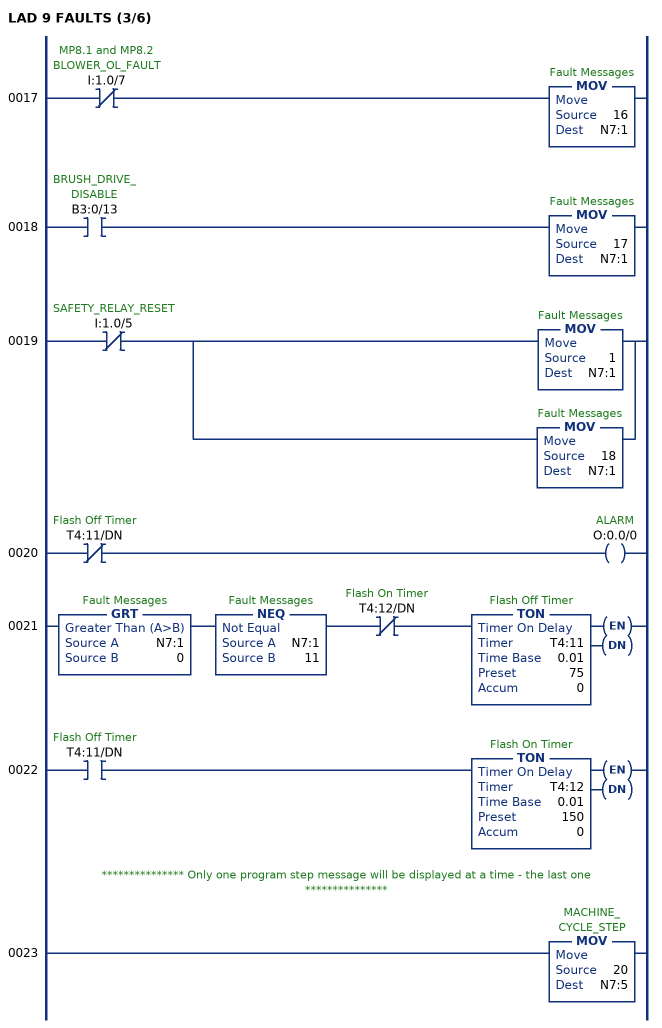
% Rung: 17 %
SOR XIO I:1.0/7 MOV 16 N7:1 EOR
%   I:1.0/7  BLOWER_OL_FAULT  "MP8.1 and MP8.2" %
%   N7:1  "Fault Messages" %
% Rung: 18 %
SOR XIC B3:0/13 MOV 17 N7:1 EOR
%   B3:0/13  BRUSH_DRIVE_DISABLE %
%   N7:1  "Fault Messages" %
% Rung: 19 %
SOR XIO I:1.0/5 BST MOV 1 N7:1 NXB MOV 18 N7:1 BND EOR
%   I:1.0/5  SAFETY_RELAY_RESET %
%   N7:1  "Fault Messages" %
% Rung: 20 %
SOR XIO T4:11/DN OTE O:0.0/0 EOR
%   T4:11  "Flash Off Timer" %
%   O:0.0/0  ALARM %
% Rung: 21 %
SOR GRT N7:1 0 NEQ N7:1 11 XIO T4:12/DN TON T4:11 0.01 75 0 EOR
%   N7:1  "Fault Messages" %
%   T4:12  "Flash On Timer" %
%   T4:11  "Flash Off Timer" %
% Rung: 22 %
SOR XIC T4:11/DN TON T4:12 0.01 150 0 EOR
%   T4:11  "Flash Off Timer" %
%   T4:12  "Flash On Timer" %
% Rung: 23 %
% *************** Only one program step message will be displayed at a time - the last one *************** %
SOR MOV 20 N7:5 EOR
%   N7:5  MACHINE_CYCLE_STEP %

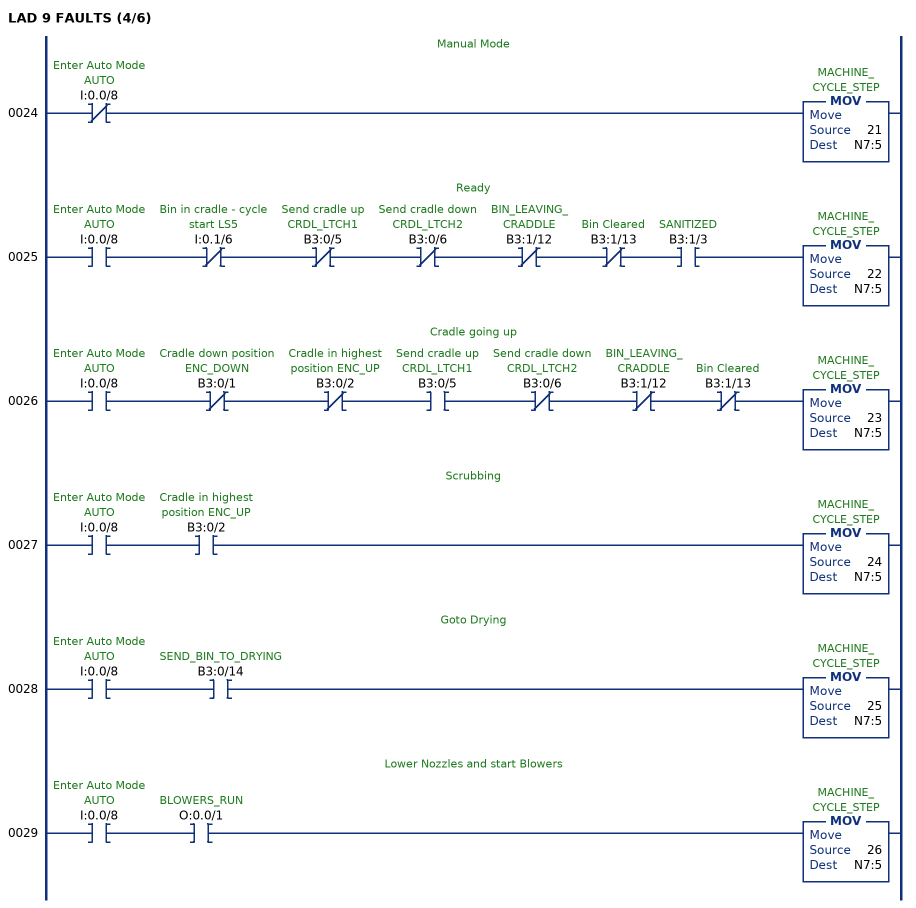
% Rung: 24 %
% Manual Mode %
SOR XIO I:0.0/8 MOV 21 N7:5 EOR
%   I:0.0/8  AUTO  "Enter Auto Mode" %
%   N7:5  MACHINE_CYCLE_STEP %
% Rung: 25 %
% Ready %
SOR XIC I:0.0/8 XIO I:0.1/6 XIO B3:0/5 XIO B3:0/6 XIO B3:1/12 XIO B3:1/13 XIC B3:1/3 MOV 22 N7:5 EOR
%   I:0.0/8  AUTO  "Enter Auto Mode" %
%   I:0.1/6  LS5  "Bin in cradle - cycle start" %
%   B3:0/5  CRDL_LTCH1  "Send cradle up" %
%   B3:0/6  CRDL_LTCH2  "Send cradle down" %
%   B3:1/12  BIN_LEAVING_CRADDLE %
%   B3:1/13  "Bin Cleared" %
%   B3:1/3  SANITIZED %
%   N7:5  MACHINE_CYCLE_STEP %
% Rung: 26 %
% Cradle going up %
SOR XIC I:0.0/8 XIO B3:0/1 XIO B3:0/2 XIC B3:0/5 XIO B3:0/6 XIO B3:1/12 XIO B3:1/13 MOV 23 N7:5 EOR
%   I:0.0/8  AUTO  "Enter Auto Mode" %
%   B3:0/1  ENC_DOWN  "Cradle down position" %
%   B3:0/2  ENC_UP  "Cradle in highest position" %
%   B3:0/5  CRDL_LTCH1  "Send cradle up" %
%   B3:0/6  CRDL_LTCH2  "Send cradle down" %
%   B3:1/12  BIN_LEAVING_CRADDLE %
%   B3:1/13  "Bin Cleared" %
%   N7:5  MACHINE_CYCLE_STEP %
% Rung: 27 %
% Scrubbing %
SOR XIC I:0.0/8 XIC B3:0/2 MOV 24 N7:5 EOR
%   I:0.0/8  AUTO  "Enter Auto Mode" %
%   B3:0/2  ENC_UP  "Cradle in highest position" %
%   N7:5  MACHINE_CYCLE_STEP %
% Rung: 28 %
% Goto Drying %
SOR XIC I:0.0/8 XIC B3:0/14 MOV 25 N7:5 EOR
%   I:0.0/8  AUTO  "Enter Auto Mode" %
%   B3:0/14  SEND_BIN_TO_DRYING %
%   N7:5  MACHINE_CYCLE_STEP %
% Rung: 29 %
% Lower Nozzles and start Blowers %
SOR XIC I:0.0/8 XIC O:0.0/1 MOV 26 N7:5 EOR
%   I:0.0/8  AUTO  "Enter Auto Mode" %
%   O:0.0/1  BLOWERS_RUN %
%   N7:5  MACHINE_CYCLE_STEP %

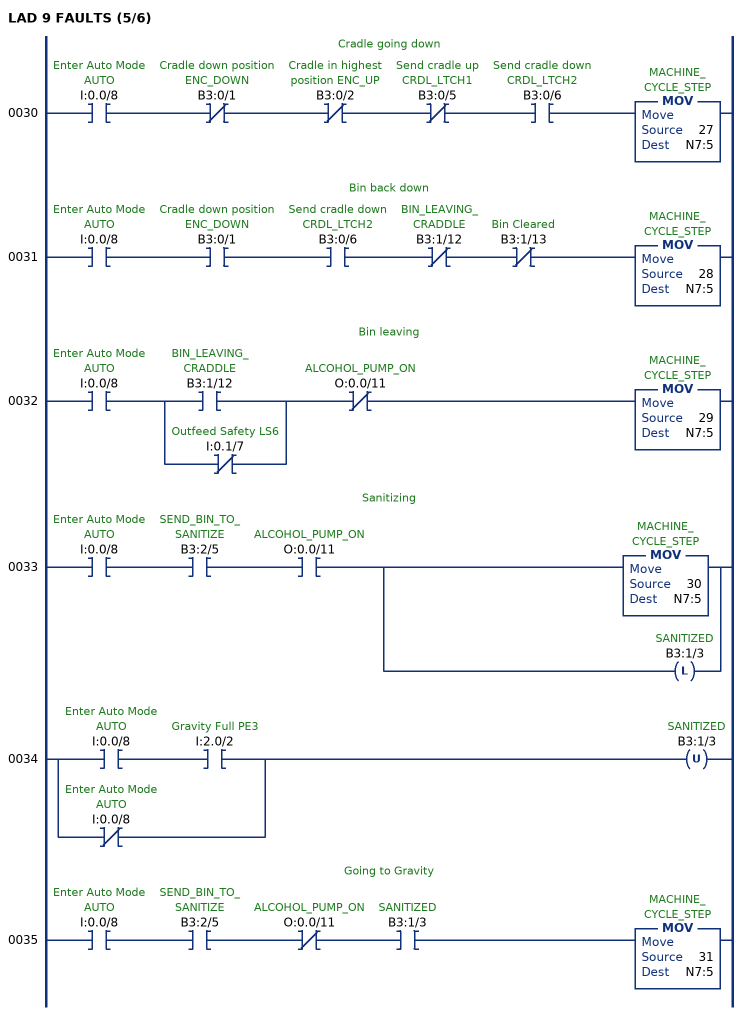
% Rung: 30 %
% Cradle going down %
SOR XIC I:0.0/8 XIO B3:0/1 XIO B3:0/2 XIO B3:0/5 XIC B3:0/6 MOV 27 N7:5 EOR
%   I:0.0/8  AUTO  "Enter Auto Mode" %
%   B3:0/1  ENC_DOWN  "Cradle down position" %
%   B3:0/2  ENC_UP  "Cradle in highest position" %
%   B3:0/5  CRDL_LTCH1  "Send cradle up" %
%   B3:0/6  CRDL_LTCH2  "Send cradle down" %
%   N7:5  MACHINE_CYCLE_STEP %
% Rung: 31 %
% Bin back down %
SOR XIC I:0.0/8 XIC B3:0/1 XIC B3:0/6 XIO B3:1/12 XIO B3:1/13 MOV 28 N7:5 EOR
%   I:0.0/8  AUTO  "Enter Auto Mode" %
%   B3:0/1  ENC_DOWN  "Cradle down position" %
%   B3:0/6  CRDL_LTCH2  "Send cradle down" %
%   B3:1/12  BIN_LEAVING_CRADDLE %
%   B3:1/13  "Bin Cleared" %
%   N7:5  MACHINE_CYCLE_STEP %
% Rung: 32 %
% Bin leaving %
SOR XIC I:0.0/8 BST XIC B3:1/12 NXB XIO I:0.1/7 BND XIO O:0.0/11 MOV 29 N7:5 EOR
%   I:0.0/8  AUTO  "Enter Auto Mode" %
%   B3:1/12  BIN_LEAVING_CRADDLE %
%   I:0.1/7  LS6  "Outfeed Safety" %
%   O:0.0/11  ALCOHOL_PUMP_ON %
%   N7:5  MACHINE_CYCLE_STEP %
% Rung: 33 %
% Sanitizing %
SOR XIC I:0.0/8 XIC B3:2/5 XIC O:0.0/11 BST MOV 30 N7:5 NXB OTL B3:1/3 BND EOR
%   I:0.0/8  AUTO  "Enter Auto Mode" %
%   B3:2/5  SEND_BIN_TO_SANITIZE %
%   O:0.0/11  ALCOHOL_PUMP_ON %
%   N7:5  MACHINE_CYCLE_STEP %
%   B3:1/3  SANITIZED %
% Rung: 34 %
SOR BST XIC I:0.0/8 XIC I:2.0/2 NXB XIO I:0.0/8 BND OTU B3:1/3 EOR
%   I:0.0/8  AUTO  "Enter Auto Mode" %
%   I:2.0/2  PE3  "Gravity Full" %
%   B3:1/3  SANITIZED %
% Rung: 35 %
% Going to Gravity %
SOR XIC I:0.0/8 XIC B3:2/5 XIO O:0.0/11 XIC B3:1/3 MOV 31 N7:5 EOR
%   I:0.0/8  AUTO  "Enter Auto Mode" %
%   B3:2/5  SEND_BIN_TO_SANITIZE %
%   O:0.0/11  ALCOHOL_PUMP_ON %
%   B3:1/3  SANITIZED %
%   N7:5  MACHINE_CYCLE_STEP %

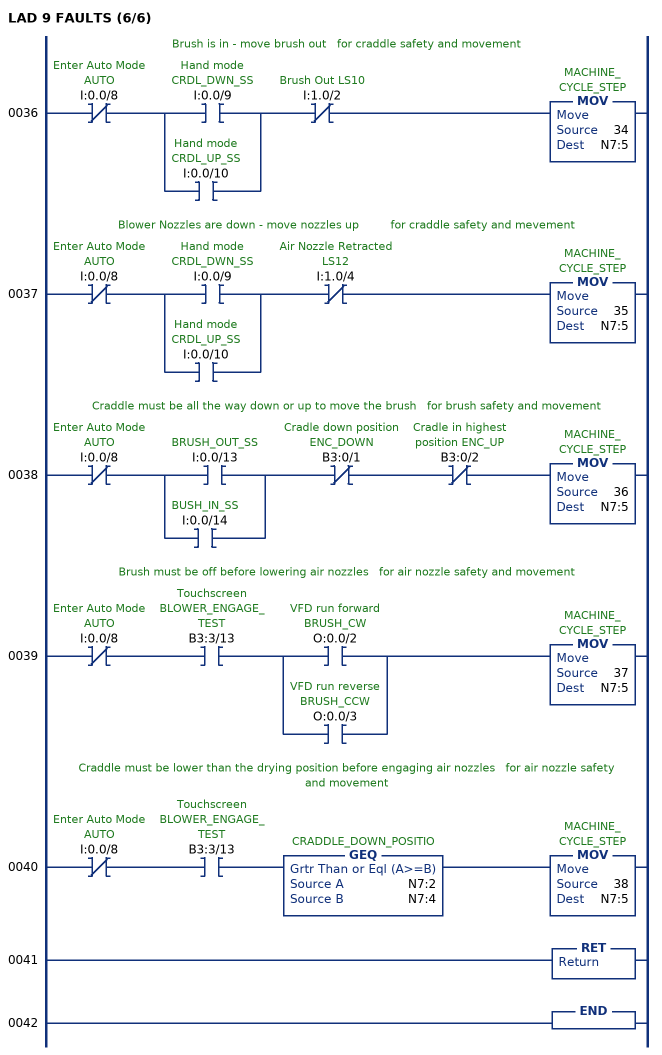
% Rung: 36 %
% Brush is in - move brush out   for craddle safety and movement %
SOR XIO I:0.0/8 BST XIC I:0.0/9 NXB XIC I:0.0/10 BND XIO I:1.0/2 MOV 34 N7:5 EOR
%   I:0.0/8  AUTO  "Enter Auto Mode" %
%   I:0.0/9  CRDL_DWN_SS  "Hand mode" %
%   I:0.0/10  CRDL_UP_SS  "Hand mode" %
%   I:1.0/2  LS10  "Brush Out" %
%   N7:5  MACHINE_CYCLE_STEP %
% Rung: 37 %
% Blower Nozzles are down - move nozzles up         for craddle safety and mevement %
SOR XIO I:0.0/8 BST XIC I:0.0/9 NXB XIC I:0.0/10 BND XIO I:1.0/4 MOV 35 N7:5 EOR
%   I:0.0/8  AUTO  "Enter Auto Mode" %
%   I:0.0/9  CRDL_DWN_SS  "Hand mode" %
%   I:0.0/10  CRDL_UP_SS  "Hand mode" %
%   I:1.0/4  LS12  "Air Nozzle Retracted" %
%   N7:5  MACHINE_CYCLE_STEP %
% Rung: 38 %
% Craddle must be all the way down or up to move the brush   for brush safety and movement %
SOR XIO I:0.0/8 BST XIC I:0.0/13 NXB XIC I:0.0/14 BND XIO B3:0/1 XIO B3:0/2 MOV 36 N7:5 EOR
%   I:0.0/8  AUTO  "Enter Auto Mode" %
%   I:0.0/13  BRUSH_OUT_SS %
%   I:0.0/14  BUSH_IN_SS %
%   B3:0/1  ENC_DOWN  "Cradle down position" %
%   B3:0/2  ENC_UP  "Cradle in highest position" %
%   N7:5  MACHINE_CYCLE_STEP %
% Rung: 39 %
% Brush must be off before lowering air nozzles   for air nozzle safety and movement %
SOR XIO I:0.0/8 XIC B3:3/13 BST XIC O:0.0/2 NXB XIC O:0.0/3 BND MOV 37 N7:5 EOR
%   I:0.0/8  AUTO  "Enter Auto Mode" %
%   B3:3/13  BLOWER_ENGAGE_TEST  "Touchscreen" %
%   O:0.0/2  BRUSH_CW  "VFD run forward" %
%   O:0.0/3  BRUSH_CCW  "VFD run reverse" %
%   N7:5  MACHINE_CYCLE_STEP %
% Rung: 40 %
% Craddle must be lower than the drying position before engaging air nozzles   for air nozzle safety and movement %
SOR XIO I:0.0/8 XIC B3:3/13 GEQ N7:2 N7:4 MOV 38 N7:5 EOR
%   I:0.0/8  AUTO  "Enter Auto Mode" %
%   B3:3/13  BLOWER_ENGAGE_TEST  "Touchscreen" %
%   N7:2  CRADDLE_DOWN_POSITIO %
%   N7:4  DRYING_POSITION %
%   N7:5  MACHINE_CYCLE_STEP %
% Rung: 41 %
SOR RET EOR
% Rung: 42 %
SOR END EOR

LADDER 10 "CONVEYORS"
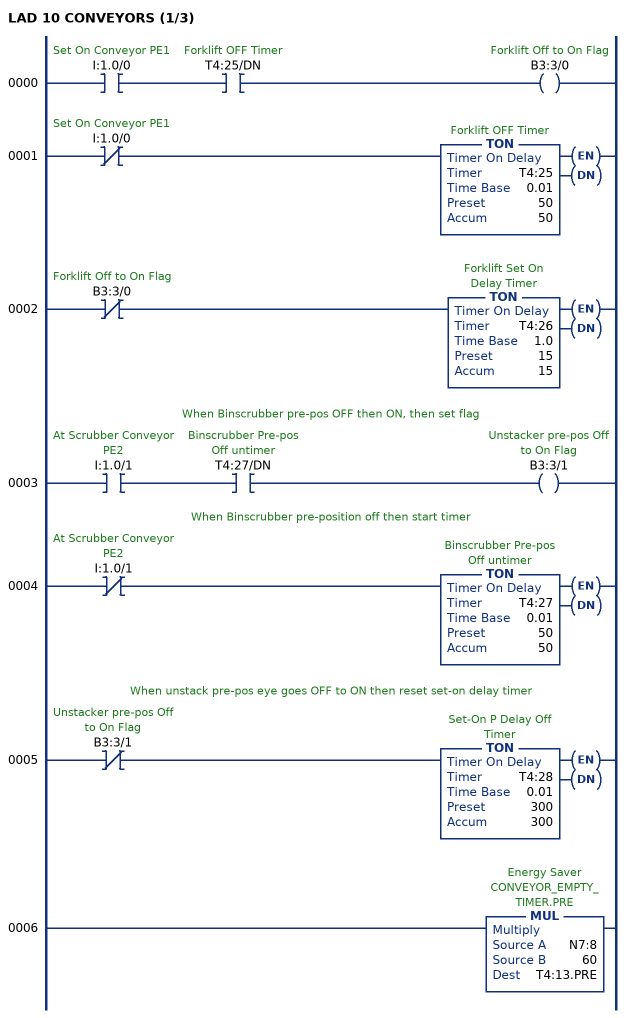
% Rung: 0 %
SOR XIC I:1.0/0 XIC T4:25/DN OTE B3:3/0 EOR
%   I:1.0/0  PE1  "Set On Conveyor" %
%   T4:25  "Forklift OFF Timer" %
%   B3:3/0  "Forklift Off to On Flag" %
% Rung: 1 %
SOR XIO I:1.0/0 TON T4:25 0.01 50 50 EOR
%   I:1.0/0  PE1  "Set On Conveyor" %
%   T4:25  "Forklift OFF Timer" %
% Rung: 2 %
SOR XIO B3:3/0 TON T4:26 1.0 15 15 EOR
%   B3:3/0  "Forklift Off to On Flag" %
%   T4:26  "Forklift Set On Delay Timer" %
% Rung: 3 %
% When Binscrubber pre-pos OFF then ON, then set flag %
SOR XIC I:1.0/1 XIC T4:27/DN OTE B3:3/1 EOR
%   I:1.0/1  PE2  "At Scrubber Conveyor" %
%   T4:27  "Binscrubber Pre-pos Off untimer" %
%   B3:3/1  "Unstacker pre-pos Off to On Flag" %
% Rung: 4 %
% When Binscrubber pre-position off then start timer %
SOR XIO I:1.0/1 TON T4:27 0.01 50 50 EOR
%   I:1.0/1  PE2  "At Scrubber Conveyor" %
%   T4:27  "Binscrubber Pre-pos Off untimer" %
% Rung: 5 %
% When unstack pre-pos eye goes OFF to ON then reset set-on delay timer %
SOR XIO B3:3/1 TON T4:28 0.01 300 300 EOR
%   B3:3/1  "Unstacker pre-pos Off to On Flag" %
%   T4:28  "Set-On P Delay Off Timer" %
% Rung: 6 %
SOR MUL N7:8 60 T4:13.PRE EOR
%   N7:8  CONVEYOR_SAVER_MINUT %
%   T4:13  CONVEYOR_EMPTY_TIMER  "Energy Saver" %

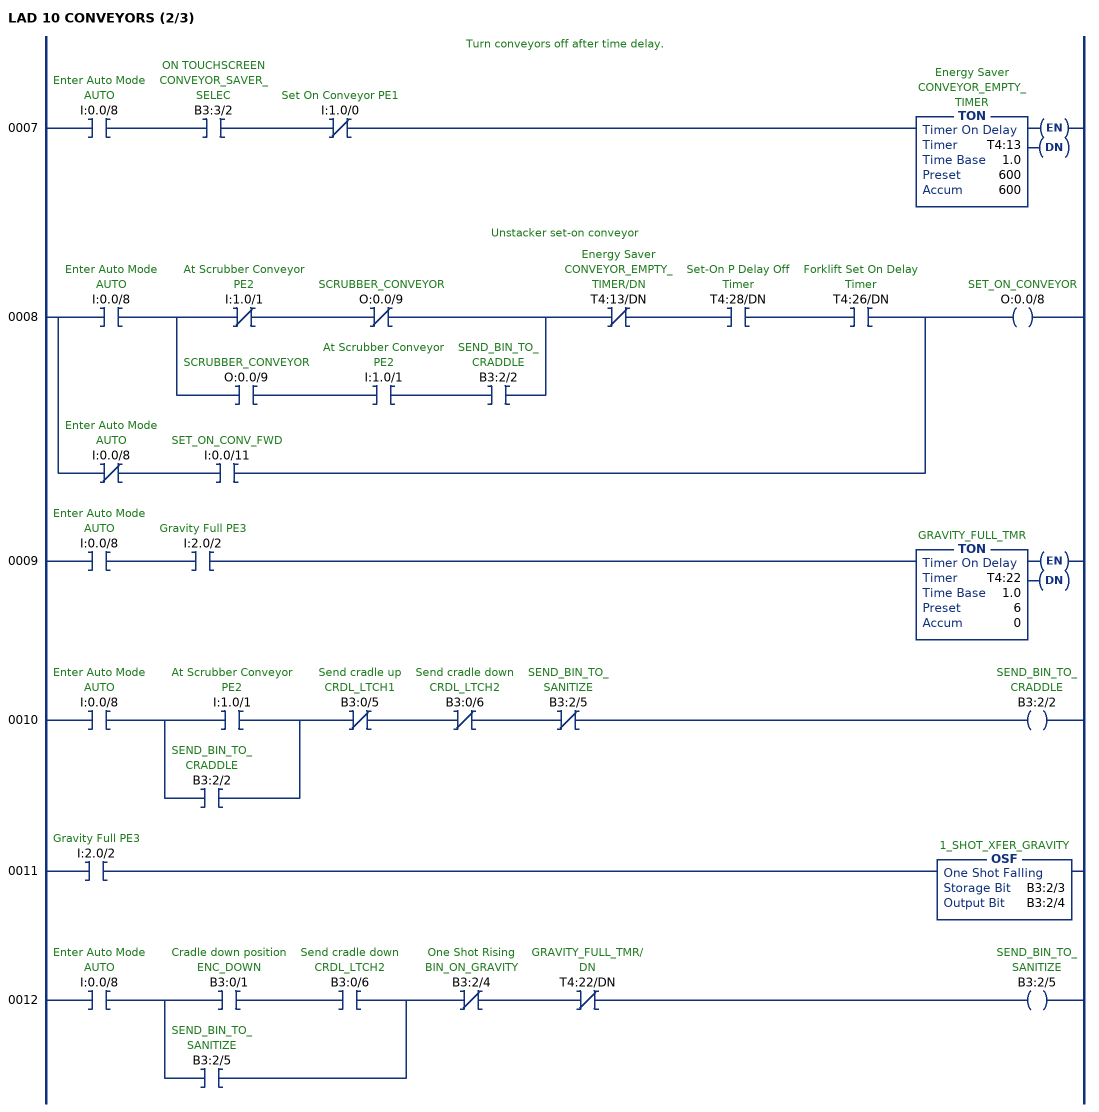
% Rung: 7 %
% Turn conveyors off after time delay. %
SOR XIC I:0.0/8 XIC B3:3/2 XIO I:1.0/0 TON T4:13 1.0 600 600 EOR
%   I:0.0/8  AUTO  "Enter Auto Mode" %
%   B3:3/2  CONVEYOR_SAVER_SELEC  "ON TOUCHSCREEN" %
%   I:1.0/0  PE1  "Set On Conveyor" %
%   T4:13  CONVEYOR_EMPTY_TIMER  "Energy Saver" %
% Rung: 8 %
% Unstacker set-on conveyor %
SOR BST XIC I:0.0/8 BST XIO I:1.0/1 XIO O:0.0/9 NXB XIC O:0.0/9 XIC I:1.0/1 XIC B3:2/2 BND XIO T4:13/DN XIC T4:28/DN XIC T4:26/DN NXB XIO I:0.0/8 XIC I:0.0/11 BND OTE O:0.0/8 EOR
%   I:0.0/8  AUTO  "Enter Auto Mode" %
%   I:1.0/1  PE2  "At Scrubber Conveyor" %
%   O:0.0/9  SCRUBBER_CONVEYOR %
%   B3:2/2  SEND_BIN_TO_CRADDLE %
%   T4:13  CONVEYOR_EMPTY_TIMER  "Energy Saver" %
%   T4:28  "Set-On P Delay Off Timer" %
%   T4:26  "Forklift Set On Delay Timer" %
%   I:0.0/11  SET_ON_CONV_FWD %
%   O:0.0/8  SET_ON_CONVEYOR %
% Rung: 9 %
SOR XIC I:0.0/8 XIC I:2.0/2 TON T4:22 1.0 6 0 EOR
%   I:0.0/8  AUTO  "Enter Auto Mode" %
%   I:2.0/2  PE3  "Gravity Full" %
%   T4:22  GRAVITY_FULL_TMR %
% Rung: 10 %
SOR XIC I:0.0/8 BST XIC I:1.0/1 NXB XIC B3:2/2 BND XIO B3:0/5 XIO B3:0/6 XIO B3:2/5 OTE B3:2/2 EOR
%   I:0.0/8  AUTO  "Enter Auto Mode" %
%   I:1.0/1  PE2  "At Scrubber Conveyor" %
%   B3:2/2  SEND_BIN_TO_CRADDLE %
%   B3:0/5  CRDL_LTCH1  "Send cradle up" %
%   B3:0/6  CRDL_LTCH2  "Send cradle down" %
%   B3:2/5  SEND_BIN_TO_SANITIZE %
% Rung: 11 %
SOR XIC I:2.0/2 OSF B3:2/3 B3:2/4 EOR
%   I:2.0/2  PE3  "Gravity Full" %
%   B3:2/3  1_SHOT_XFER_GRAVITY %
%   B3:2/4  BIN_ON_GRAVITY  "One Shot Rising" %
% Rung: 12 %
SOR XIC I:0.0/8 BST XIC B3:0/1 XIC B3:0/6 NXB XIC B3:2/5 BND XIO B3:2/4 XIO T4:22/DN OTE B3:2/5 EOR
%   I:0.0/8  AUTO  "Enter Auto Mode" %
%   B3:0/1  ENC_DOWN  "Cradle down position" %
%   B3:0/6  CRDL_LTCH2  "Send cradle down" %
%   B3:2/5  SEND_BIN_TO_SANITIZE %
%   B3:2/4  BIN_ON_GRAVITY  "One Shot Rising" %
%   T4:22  GRAVITY_FULL_TMR %

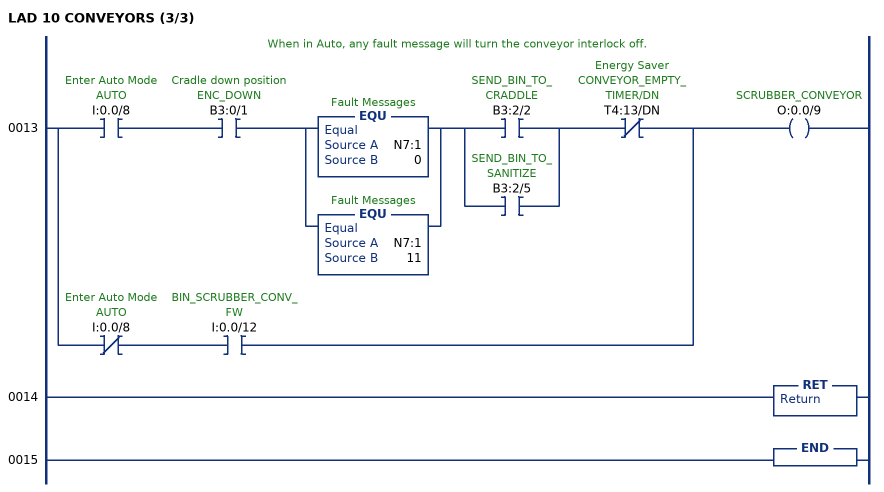
% Rung: 13 %
% When in Auto, any fault message will turn the conveyor interlock off. %
SOR BST XIC I:0.0/8 XIC B3:0/1 BST EQU N7:1 0 NXB EQU N7:1 11 BND BST XIC B3:2/2 NXB XIC B3:2/5 BND XIO T4:13/DN NXB XIO I:0.0/8 XIC I:0.0/12 BND OTE O:0.0/9 EOR
%   I:0.0/8  AUTO  "Enter Auto Mode" %
%   B3:0/1  ENC_DOWN  "Cradle down position" %
%   N7:1  "Fault Messages" %
%   B3:2/2  SEND_BIN_TO_CRADDLE %
%   B3:2/5  SEND_BIN_TO_SANITIZE %
%   T4:13  CONVEYOR_EMPTY_TIMER  "Energy Saver" %
%   I:0.0/12  BIN_SCRUBBER_CONV_FW %
%   O:0.0/9  SCRUBBER_CONVEYOR %
% Rung: 14 %
SOR RET EOR
% Rung: 15 %
SOR END EOR

LADDER 11 "BIN SIZING"
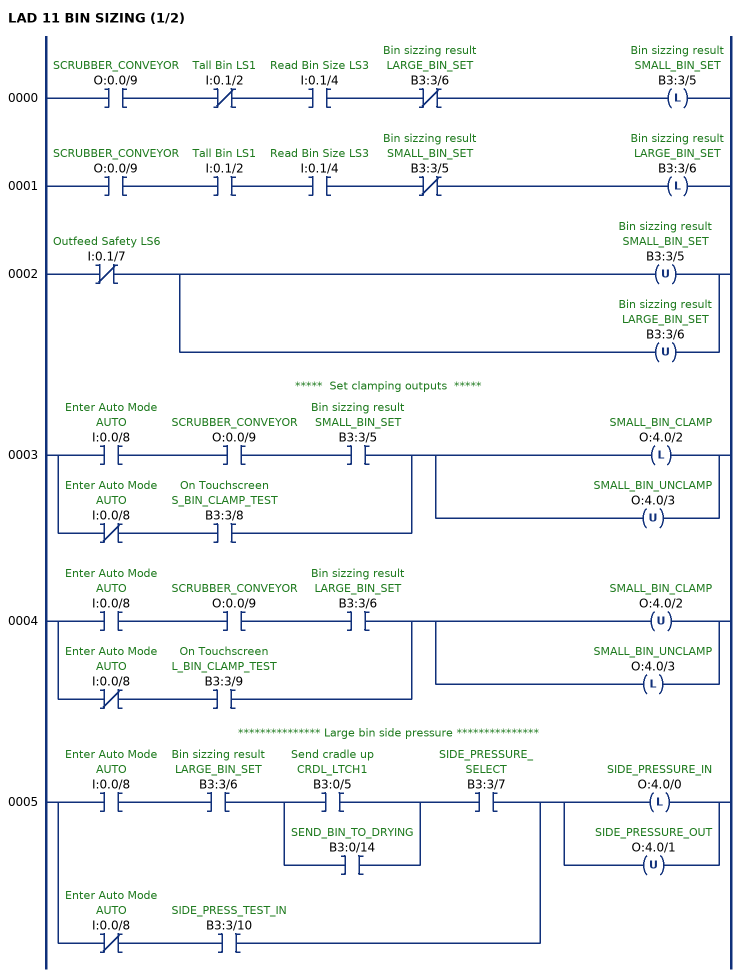
% Rung: 0 %
SOR XIC O:0.0/9 XIO I:0.1/2 XIC I:0.1/4 XIO B3:3/6 OTL B3:3/5 EOR
%   O:0.0/9  SCRUBBER_CONVEYOR %
%   I:0.1/2  LS1  "Tall Bin" %
%   I:0.1/4  LS3  "Read Bin Size" %
%   B3:3/6  LARGE_BIN_SET  "Bin sizzing result" %
%   B3:3/5  SMALL_BIN_SET  "Bin sizzing result" %
% Rung: 1 %
SOR XIC O:0.0/9 XIC I:0.1/2 XIC I:0.1/4 XIO B3:3/5 OTL B3:3/6 EOR
%   O:0.0/9  SCRUBBER_CONVEYOR %
%   I:0.1/2  LS1  "Tall Bin" %
%   I:0.1/4  LS3  "Read Bin Size" %
%   B3:3/5  SMALL_BIN_SET  "Bin sizzing result" %
%   B3:3/6  LARGE_BIN_SET  "Bin sizzing result" %
% Rung: 2 %
SOR XIO I:0.1/7 BST OTU B3:3/5 NXB OTU B3:3/6 BND EOR
%   I:0.1/7  LS6  "Outfeed Safety" %
%   B3:3/5  SMALL_BIN_SET  "Bin sizzing result" %
%   B3:3/6  LARGE_BIN_SET  "Bin sizzing result" %
% Rung: 3 %
% *****  Set clamping outputs  ***** %
SOR BST XIC I:0.0/8 XIC O:0.0/9 XIC B3:3/5 NXB XIO I:0.0/8 XIC B3:3/8 BND BST OTL O:4.0/2 NXB OTU O:4.0/3 BND EOR
%   I:0.0/8  AUTO  "Enter Auto Mode" %
%   O:0.0/9  SCRUBBER_CONVEYOR %
%   B3:3/5  SMALL_BIN_SET  "Bin sizzing result" %
%   B3:3/8  S_BIN_CLAMP_TEST  "On Touchscreen" %
%   O:4.0/2  SMALL_BIN_CLAMP %
%   O:4.0/3  SMALL_BIN_UNCLAMP %
% Rung: 4 %
SOR BST XIC I:0.0/8 XIC O:0.0/9 XIC B3:3/6 NXB XIO I:0.0/8 XIC B3:3/9 BND BST OTU O:4.0/2 NXB OTL O:4.0/3 BND EOR
%   I:0.0/8  AUTO  "Enter Auto Mode" %
%   O:0.0/9  SCRUBBER_CONVEYOR %
%   B3:3/6  LARGE_BIN_SET  "Bin sizzing result" %
%   B3:3/9  L_BIN_CLAMP_TEST  "On Touchscreen" %
%   O:4.0/2  SMALL_BIN_CLAMP %
%   O:4.0/3  SMALL_BIN_UNCLAMP %
% Rung: 5 %
% *************** Large bin side pressure *************** %
SOR BST XIC I:0.0/8 XIC B3:3/6 BST XIC B3:0/5 NXB XIC B3:0/14 BND XIC B3:3/7 NXB XIO I:0.0/8 XIC B3:3/10 BND BST OTL O:4.0/0 NXB OTU O:4.0/1 BND EOR
%   I:0.0/8  AUTO  "Enter Auto Mode" %
%   B3:3/6  LARGE_BIN_SET  "Bin sizzing result" %
%   B3:0/5  CRDL_LTCH1  "Send cradle up" %
%   B3:0/14  SEND_BIN_TO_DRYING %
%   B3:3/7  SIDE_PRESSURE_SELECT %
%   B3:3/10  SIDE_PRESS_TEST_IN %
%   O:4.0/0  SIDE_PRESSURE_IN %
%   O:4.0/1  SIDE_PRESSURE_OUT %

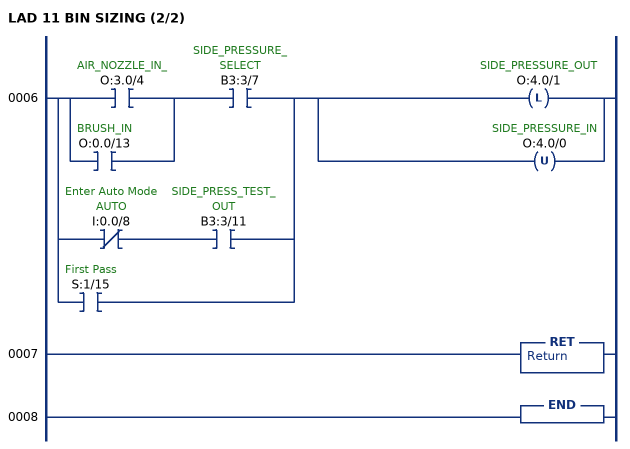
% Rung: 6 %
SOR BST BST BST XIC O:3.0/4 NXB XIC O:0.0/13 BND XIC B3:3/7 NXB XIO I:0.0/8 XIC B3:3/11 BND NXB XIC S:1/15 BND BST OTL O:4.0/1 NXB OTU O:4.0/0 BND EOR
%   O:3.0/4  AIR_NOZZLE_IN_ %
%   O:0.0/13  BRUSH_IN %
%   B3:3/7  SIDE_PRESSURE_SELECT %
%   I:0.0/8  AUTO  "Enter Auto Mode" %
%   B3:3/11  SIDE_PRESS_TEST_OUT %
%   S:1/15  "First Pass" %
%   O:4.0/1  SIDE_PRESSURE_OUT %
%   O:4.0/0  SIDE_PRESSURE_IN %
% Rung: 7 %
SOR RET EOR
% Rung: 8 %
SOR END EOR

OTHER DOCUMENTED ADDRESSES
  B3:1/9  SPARE_TC
  B3:2/14  DRYING_POS_REACHED
  B3:2/15  DRYING_COMPLETED
  B3:4/3  RELEASE_FOR_SANITIZE
  B3:4/11  INNER_NOZZLE_TMR_BIT
  C5:0/CU  EVENT_COUNTER
  I:0.1/3  SPARE1
  I:1.0/10  "Set-On Forklift"
  I:1.0/11  "De-stack Approach"
  I:1.0/13  "De-stacker Stack In"
  I:1.0/15  "De-stacker Dogs Out"
  I:2.0/3  PS2_ALCOHOL
  L10:1/1  FAULT_MESSAGES
  N7:1/0  "Fault-Infeed Blocked"
  N7:1/1  "Fault-Outfeed Blocked"
  N7:1/2  "Fault-Cradle Overtravel Up"
  N7:1/3  "Fault-Cradle Overtravel down"
  N7:1/4  "Fault-Torque Cradle Inverter"
  N7:1/5  "Main Tank Low"
  N7:1/6  "Encoder Fault"
  N7:1/7  "Fill Main Tank"
  N7:7  LOWER_WASH_TURN_OFF
  N7:14  TALL_BIN_PREWASH
  N9:0  K1
  O:0.0/7  NOT_USED
  T4:0/EN  CRDL_DWN_T  "Allows cradle to set down completely before conv starts"
  T4:1  CRDL_FLT_T1
  T4:2  CRDL_FLT_T2
  T4:6  SANITIZE_T
  T4:7  CRDL_DWN_T2  "Inhibits cradle up for 5 sec. after cradle sets down"
  T4:10  CRADLE_TIMER  "Cradle travel watch dog timer"
  T4:16  CRADLE_DOWN_TIMER

COMMENTS NOT ATTACHED TO A CURRENT RUNG
  N7:1/0: As long as the bit is set, the message will be displayed.  Bit #1 is Message #1.  Bit #3 is message #4.  Binary to decimal.
  T4:6.PRE: As long as the bit is set, the message will be displayed.  Bit #1 is Message #1.  Bit #3 is message #4.  Binary to decimal.
  T4:7: Timer not used
  B3:4/4: ***************  Sanitize ***************
  N7:9: Change minutes to seconds for the timer
  T4:19: Prewash delay for large bins

REVISION NOTES
  0: Added barrier and overtravel tatches
  1: Added indepentent barrier and overtravel catches
  2: Changed ffrom Panel #8.  Added B3:0/1 to prevent B3:0/5 from latching up while cradle is not down
  3: Added more troubleshooting help - step sequences
  4: Costa Rica Panel #19 with individual upper and lower wash solenoids

DATA TABLE (non-zero values as saved)
DATA B3
% B3:0 % 0X015A 0X0800 0X0420 0X00C4 0X0101
DATA T4
% .PRE .ACC %
% T4:0 % 50 50
% T4:1 % 1 0
% T4:2 % 1 0
% T4:3 % 500 0
% T4:4 % 2 2
% T4:5 % 5 0
% T4:6 % 658 0
% T4:7 % 375 500
% T4:8 % 5 0
% T4:9 % 2 2
% T4:10 % 500 0
% T4:11 % 75 0
% T4:12 % 150 0
% T4:13 % 600 600
% T4:14 % 10 0
% T4:15 % 6 0
% T4:16 % 6 0
% T4:17 % 10 0
% T4:18 % 100 0
% T4:19 % 5 0
% T4:20 % 1 0
% T4:21 % 150 0
% T4:22 % 6 0
% T4:23 % 400 0
% T4:24 % 1 0
% T4:25 % 50 50
% T4:26 % 15 15
% T4:27 % 50 50
% T4:28 % 300 300
% T4:29 % 600 600
% T4:30 % 5 0
% T4:31 % 1 0
% T4:32 % 1 0
% T4:33 % 1 0
DATA N7
% N7:0 % 86 11 10 55 106 31 27 0 10 0
% N7:10 % 5 5 10 10 0 0 1 238 10 0
% N7:20 % 10 12 141 105 45 0 1 1 10 10
DATA F8
% F8:0 % 18
